// TIA Portal V20 export
FUNCTION "EM5_TeachingData" : Void   // FC85, LAD
// stored: Namespace Unit1.Em5, SetENOAutomatically false
BEGIN

REGION Network 2 (SCL): Transfer PnP Left AxisX Teaching Position
   // Transfer PnP Left AxisX Position 0
   "Unit1.Em5.HmiInterface".cmTransferPnPLeftAxisX.configuration.setPositions[0].position := 107.84;
   "Unit1.Em5.HmiInterface".cmTransferPnPLeftAxisX.configuration.setPositions[0].velocity := 50.0;

   // Transfer PnP Left AxisX Position 1
   "Unit1.Em5.HmiInterface".cmTransferPnPLeftAxisX.configuration.setPositions[1].position := 107.84;
   "Unit1.Em5.HmiInterface".cmTransferPnPLeftAxisX.configuration.setPositions[1].velocity := 50.0;

   // Transfer PnP Left AxisX Position 2
   "Unit1.Em5.HmiInterface".cmTransferPnPLeftAxisX.configuration.setPositions[2].position := 1064.0;
   "Unit1.Em5.HmiInterface".cmTransferPnPLeftAxisX.configuration.setPositions[2].velocity := 50.0;

   // Transfer PnP Left AxisX Position 3
   "Unit1.Em5.HmiInterface".cmTransferPnPLeftAxisX.configuration.setPositions[3].position := 1712.0;
   "Unit1.Em5.HmiInterface".cmTransferPnPLeftAxisX.configuration.setPositions[3].velocity := 50.0;

   // Transfer PnP Left AxisX Position 4
   "Unit1.Em5.HmiInterface".cmTransferPnPLeftAxisX.configuration.setPositions[4].position := 2366.7;
   "Unit1.Em5.HmiInterface".cmTransferPnPLeftAxisX.configuration.setPositions[4].velocity := 50.0;


   //////////////////////// ZONE ///////////////////////
   "Unit1.Em5.HmiInterface".cmTransferPnPLeftAxisX.configuration.setPositions[9].position := 107.84;
   "Unit1.Em5.HmiInterface".cmTransferPnPLeftAxisX.configuration.setPositions[9].velocity := 50.0;
END_REGION

REGION Network 3 (SCL): Transfer PnP Left AxisY Teaching Position
   // Transfer PnP Left AxisY Position 0
   "Unit1.Em5.HmiInterface".cmTransferPnPLeftAxisY.configuration.setPositions[0].position := 0.0;
   "Unit1.Em5.HmiInterface".cmTransferPnPLeftAxisY.configuration.setPositions[0].velocity := 10.0;

   // Transfer PnP Left AxisY Position 1
   "Unit1.Em5.HmiInterface".cmTransferPnPLeftAxisY.configuration.setPositions[1].position := 480.0;
   "Unit1.Em5.HmiInterface".cmTransferPnPLeftAxisY.configuration.setPositions[1].velocity := 10.0;

   // Transfer PnP Left AxisY Position 2
   "Unit1.Em5.HmiInterface".cmTransferPnPLeftAxisY.configuration.setPositions[2].position := 482.0;
   "Unit1.Em5.HmiInterface".cmTransferPnPLeftAxisY.configuration.setPositions[2].velocity := 10.0;

   // Transfer PnP Left AxisY Position 3
   "Unit1.Em5.HmiInterface".cmTransferPnPLeftAxisY.configuration.setPositions[3].position := 482.0;
   "Unit1.Em5.HmiInterface".cmTransferPnPLeftAxisY.configuration.setPositions[3].velocity := 10.0;

   // Transfer PnP Left AxisY Position 4
   "Unit1.Em5.HmiInterface".cmTransferPnPLeftAxisY.configuration.setPositions[4].position := 471.0;
   "Unit1.Em5.HmiInterface".cmTransferPnPLeftAxisY.configuration.setPositions[4].velocity := 10.0;
END_REGION

REGION Network 4 (SCL): Transfer PnP Left AxisZ Teaching Position
   // Transfer PnP Left AxisZ Position 0
   "Unit1.Em5.HmiInterface".cmTransferPnPLeftAxisZ.configuration.setPositions[0].position := 15.5;
   "Unit1.Em5.HmiInterface".cmTransferPnPLeftAxisZ.configuration.setPositions[0].velocity := 10.0;

   // Transfer PnP Left AxisZ Position 1
   "Unit1.Em5.HmiInterface".cmTransferPnPLeftAxisZ.configuration.setPositions[1].position := 15.5;
   "Unit1.Em5.HmiInterface".cmTransferPnPLeftAxisZ.configuration.setPositions[1].velocity := 10.0;

   // Transfer PnP Left AxisZ Position 2
   "Unit1.Em5.HmiInterface".cmTransferPnPLeftAxisZ.configuration.setPositions[2].position := 78.59;
   "Unit1.Em5.HmiInterface".cmTransferPnPLeftAxisZ.configuration.setPositions[2].velocity := 10.0;

   // Transfer PnP Left AxisZ Position 3
   "Unit1.Em5.HmiInterface".cmTransferPnPLeftAxisZ.configuration.setPositions[3].position := 78.59;
   "Unit1.Em5.HmiInterface".cmTransferPnPLeftAxisZ.configuration.setPositions[3].velocity := 10.0;

   // Transfer PnP Left AxisZ Position 4
   "Unit1.Em5.HmiInterface".cmTransferPnPLeftAxisZ.configuration.setPositions[4].position := 100.2;
   "Unit1.Em5.HmiInterface".cmTransferPnPLeftAxisZ.configuration.setPositions[4].velocity := 10.0;
END_REGION

REGION Network 5 (SCL): Transfer PnP Right AxisX Teaching Position
   // Transfer PnP Right AxisX Position 0
   "Unit1.Em5.HmiInterface".cmTransferPnPRightAxisX.configuration.setPositions[0].position := 1250.0;
   "Unit1.Em5.HmiInterface".cmTransferPnPRightAxisX.configuration.setPositions[0].velocity := 50.0;

   // Transfer PnP Right AxisX Position 1
   "Unit1.Em5.HmiInterface".cmTransferPnPRightAxisX.configuration.setPositions[1].position := 101.4;
   "Unit1.Em5.HmiInterface".cmTransferPnPRightAxisX.configuration.setPositions[1].velocity := 50.0;

   // Transfer PnP Right AxisX Position 2
   "Unit1.Em5.HmiInterface".cmTransferPnPRightAxisX.configuration.setPositions[2].position := 719.5;
   "Unit1.Em5.HmiInterface".cmTransferPnPRightAxisX.configuration.setPositions[2].velocity := 50.0;

   // Transfer PnP Right AxisX Position 3
   "Unit1.Em5.HmiInterface".cmTransferPnPRightAxisX.configuration.setPositions[3].position := 1250.0;
   "Unit1.Em5.HmiInterface".cmTransferPnPRightAxisX.configuration.setPositions[3].velocity := 50.0;

   // Transfer PnP Right AxisX Position 4
   "Unit1.Em5.HmiInterface".cmTransferPnPRightAxisX.configuration.setPositions[4].position := 1871.0;
   "Unit1.Em5.HmiInterface".cmTransferPnPRightAxisX.configuration.setPositions[4].velocity := 50.0;
END_REGION

REGION Network 6 (SCL): Transfer PnP Right AxisY Teaching Position
   // Transfer PnP Right AxisY Position 0
   "Unit1.Em5.HmiInterface".cmTransferPnPRightAxisY.configuration.setPositions[0].position := 14.0;
   "Unit1.Em5.HmiInterface".cmTransferPnPRightAxisY.configuration.setPositions[0].velocity := 10.0;

   // Transfer PnP Right AxisY Position 1
   "Unit1.Em5.HmiInterface".cmTransferPnPRightAxisY.configuration.setPositions[1].position := 491.0;
   "Unit1.Em5.HmiInterface".cmTransferPnPRightAxisY.configuration.setPositions[1].velocity := 10.0;

   // Transfer PnP Right AxisY Position 2
   "Unit1.Em5.HmiInterface".cmTransferPnPRightAxisY.configuration.setPositions[2].position := 471.0;
   "Unit1.Em5.HmiInterface".cmTransferPnPRightAxisY.configuration.setPositions[2].velocity := 10.0;

   // Transfer PnP Right AxisY Position 3
   "Unit1.Em5.HmiInterface".cmTransferPnPRightAxisY.configuration.setPositions[3].position := 461.0;
   "Unit1.Em5.HmiInterface".cmTransferPnPRightAxisY.configuration.setPositions[3].velocity := 10.0;

   // Transfer PnP Right AxisY Position 4
   "Unit1.Em5.HmiInterface".cmTransferPnPRightAxisY.configuration.setPositions[4].position := 467.0;
   "Unit1.Em5.HmiInterface".cmTransferPnPRightAxisY.configuration.setPositions[4].velocity := 10.0;


   //////////////////////// ZONE ///////////////////////
   "Unit1.Em5.HmiInterface".cmTransferPnPRightAxisX.configuration.setPositions[8].position := 14.84;
   "Unit1.Em5.HmiInterface".cmTransferPnPRightAxisX.configuration.setPositions[8].velocity := 10.0;
END_REGION

REGION Network 7 (SCL): Transfer PnP Right AxisZ Teaching Position
   // Transfer PnP Right AxisZ Position 0
   "Unit1.Em5.HmiInterface".cmTransferPnPRightAxisZ.configuration.setPositions[0].position := 75.3;
   "Unit1.Em5.HmiInterface".cmTransferPnPRightAxisZ.configuration.setPositions[0].velocity := 10.0;

   // Transfer PnP Right AxisZ Position 1
   "Unit1.Em5.HmiInterface".cmTransferPnPRightAxisZ.configuration.setPositions[1].position := 75.3;
   "Unit1.Em5.HmiInterface".cmTransferPnPRightAxisZ.configuration.setPositions[1].velocity := 10.0;

   // Transfer PnP Right AxisZ Position 2
   "Unit1.Em5.HmiInterface".cmTransferPnPRightAxisZ.configuration.setPositions[2].position := 78.5;
   "Unit1.Em5.HmiInterface".cmTransferPnPRightAxisZ.configuration.setPositions[2].velocity := 10.0;

   // Transfer PnP Right AxisZ Position 3
   "Unit1.Em5.HmiInterface".cmTransferPnPRightAxisZ.configuration.setPositions[3].position := 77.04;
   "Unit1.Em5.HmiInterface".cmTransferPnPRightAxisZ.configuration.setPositions[3].velocity := 10.0;

   // Transfer PnP Right AxisZ Position 4
   "Unit1.Em5.HmiInterface".cmTransferPnPRightAxisZ.configuration.setPositions[4].position := 104.0;
   "Unit1.Em5.HmiInterface".cmTransferPnPRightAxisZ.configuration.setPositions[4].velocity := 10.0;

   // Transfer PnP Right AxisZ Position 5
   "Unit1.Em5.HmiInterface".cmTransferPnPRightAxisZ.configuration.setPositions[4].position := 121.0;
   "Unit1.Em5.HmiInterface".cmTransferPnPRightAxisZ.configuration.setPositions[4].velocity := 10.0;
END_REGION
END_FUNCTION
